Staubli VAL3: TRAJ.dtx

public num distance
public num moveType = 1
public num nFrameIndex
public num nGasPressure = 90
public num nIndexGun = 1
public num nLaserPower = 60
public num nPWMPercent = 100
public num nStop
public num nTcpAction
public num nTime
public num nJointMode = 1
public string comment = "moveL"
public string instruction
public bool toStop
public frame fTrack = {fatherId=world[0]}
public pointRx pCircle = {fatherId=fTrack[0]}
public pointRx pO = {fatherId=world[0]}
public pointRx pX = {fatherId=world[0]}
public pointRx pY = {fatherId=world[0]}
public pointRx points = {wrist=wfree, fatherId=fTrack[0]}
public mdesc nom_speed = {accel=7.5, vel=50, decel=7.5, tmax=100, rmax=600, leave=1, reach=1}
